{attribute 'GeneratedUsingTerminal: EK1122-0000-0018'}
{attribute addProperty BoxType "EK1122-0000-0018"}
{attribute addProperty Id "Term_17_EK1100Term_17_EK1100_DA855F56140"}
{attribute addProperty CRC "1697508353"}
{attribute addProperty Size "140"}
TYPE Term_16_EK1122_652DEC01 EXTENDS EK1122_1FC0878B :
STRUCT
	{attribute addProperty Name "Term_17_EK1100"}
	{attribute addProperty PreviousPort "Term 16 (EK1122) : D"}
	Term_17_EK1100 : Term_17_EK1100_DA855F56;
END_STRUCT
END_TYPE

(* stored: Version 1.2.0.0, ProductVersion 3.1.4024.9
   DUT Term_16_EK1122_652DEC01: Id {4db9f89a-ab3a-03d9-1b63-4df49bd0020b} *)
